{attribute 'qualified_only'}
{attribute 'strict'}
TYPE E_Light :
(
	green,
	Red
);
END_TYPE

(* stored: Version 1.1.0.1, ProductVersion 3.1.4024.9
   DUT E_Light: Id {9a6de14f-db84-47f0-b62e-e52227db1606} *)
